FUNCTION_BLOCK ACMethodRouteBase EXTENDS ACMethodBase IMPLEMENTS IACMethodRouteBase
VAR_INPUT
END_VAR
VAR_OUTPUT
END_VAR
VAR
END_VAR
VAR PERSISTENT
	_Route : PARoute;
END_VAR

METHOD PUBLIC AssignRoute : BOOL
VAR_INPUT
	iAssignWithFunction : IPAProcessFunction;
END_VAR
VAR
	i : INT;
	iControlModule : IPAControlModule;
END_VAR
IF NOT _Route._IsResolved THEN
	AssignRoute := FALSE;
	RETURN;
END_IF

// TODO: Wegwechsel einbauen bzw. aktualsiierung der Route vom Client aus?

// Prüfe zuerst ob alle Stuerungsmodule nicht belegt sind
FOR i:=1 TO GCL.cRouteItemMAX BY 1
  DO    
  	IF _Route._Items[i] <> 0 THEN
		IF __QUERYINTERFACE(_Route._Items[i].Source.Parent, iControlModule) THEN
			IF iControlModule.AllocatedByWay THEN
				AssignRoute := FALSE;
				RETURN;				
			END_IF
		END_IF
		IF __QUERYINTERFACE(_Route._Items[i].Target.Parent, iControlModule) THEN
			IF iControlModule.AllocatedByWay THEN
				AssignRoute := FALSE;
				RETURN;				
			END_IF
		END_IF
	END_IF
  	_Route._Items[i] := 0;
END_FOR;

// Setze Belegung durch diese Funktion
FOR i:=1 TO GCL.cRouteItemMAX BY 1
  DO    
  	IF _Route._Items[i] <> 0 THEN
		IF __QUERYINTERFACE(_Route._Items[i].Source.Parent, iControlModule) THEN
			iControlModule.AllocatedByFunction := iAssignWithFunction;
		END_IF
		IF __QUERYINTERFACE(_Route._Items[i].Target.Parent, iControlModule) THEN
			iControlModule.AllocatedByFunction := iAssignWithFunction;
		END_IF
		_Route._Items[i].AllocatedByFunction := iAssignWithFunction;
	END_IF
END_FOR;
_Route._IsAssigned := TRUE;
END_METHOD

PROPERTY PUBLIC FirstCModuleInRoute : IPAControlModule
GET
VAR
	i : INT;
	iControlModule : IPAControlModule;
END_VAR
FOR i:=1 TO GCL.cRouteItemMAX BY 1
  DO    
  	IF _Route._Items[i] <> 0 THEN
		IF __QUERYINTERFACE(_Route._Items[i].Source.Parent, iControlModule) THEN
			FirstCModuleInRoute := iControlModule;
			RETURN;
		END_IF
	END_IF
END_FOR;
FirstCModuleInRoute := 0;
END_GET
END_PROPERTY

PROPERTY PUBLIC LastCModuleInRoute : IPAControlModule
GET
VAR
	i : INT;
	iControlModule : IPAControlModule;
	iLastCModule : IPAControlModule;
END_VAR
iLastCModule := 0;
FOR i:=1 TO GCL.cRouteItemMAX BY 1
  DO    
  	IF _Route._Items[i] <> 0 THEN
		IF __QUERYINTERFACE(_Route._Items[i].Target.Parent, iControlModule) THEN
			iLastCModule := iControlModule;
			RETURN;
		END_IF
	ELSE
		EXIT;
	END_IF
END_FOR;
LastCModuleInRoute := iLastCModule;
END_GET
END_PROPERTY

METHOD PUBLIC ResetRoute
VAR_INPUT
END_VAR
VAR
	i : INT;
	iControlModule : IPAControlModule;
END_VAR
IF NOT _Route._IsResolved AND NOT _Route._IsAssigned THEN
	RETURN;
END_IF
FOR i:=1 TO GCL.cRouteItemMAX BY 1
  DO    
  	// Lösche Wegebelegung auf den Steuerungsmodulen
  	IF  _Route._Items[i] <> 0 THEN
		IF __QUERYINTERFACE(_Route._Items[i].Source.Parent, iControlModule) THEN
			iControlModule.AllocatedByFunction := 0;
		END_IF
		IF __QUERYINTERFACE(_Route._Items[i].Target.Parent, iControlModule) THEN
			iControlModule.AllocatedByFunction := 0;
		END_IF
	END_IF
  	_Route._Items[i] := 0;
END_FOR;
_Route._IsResolved := FALSE;
_Route._IsAssigned := FALSE;
END_METHOD

METHOD PUBLIC ResolveRoutePointers : BOOL
VAR_INPUT
	routeToResolve : PARoutePointers;	
	parentComp : IACComponent;
END_VAR
VAR
	i: INT;
	pEdge : IACEdge;
	pEdgeToTest : IACObject;
END_VAR
FOR i:=1 TO GCL.cRouteItemMAX BY 1
  DO
  	_Route._Items[i] := 0;
	IF routeToResolve._InstanceID[i] = 0 THEN
		CONTINUE;
	END_IF
	pEdgeToTest := parentComp.FindObjectByID(routeToResolve._InstanceID[i]);
	IF pEdgeToTest = 0 AND __QUERYINTERFACE(pEdgeToTest, pEdge) THEN
		_Route._Items[i] := pEdge;		
	END_IF
END_FOR;
_Route._IsResolved := TRUE;
END_METHOD

PROPERTY PUBLIC Route : PARoute
GET
Route := _Route;
END_GET
END_PROPERTY

END_FUNCTION_BLOCK

(* stored: Version 1.1.0.1, ProductVersion 3.1.4022.7
   POU ACMethodRouteBase: Id {f92ea2b6-0103-4083-9ec7-d643bb944132}, SpecialFunc None
   Method AssignRoute: Id {03406dd0-2b2c-455a-a85a-47dc4bd5e337}
   Property FirstCModuleInRoute: Id {27162ce5-5620-431d-b7a8-f2b257fbb57d}
   Get Get: Id {d437d142-8ff9-4378-b40e-0aa4bb72caa1}
   Property LastCModuleInRoute: Id {6fd6225f-b074-457f-988b-c05b459db755}
   Get Get: Id {3a094643-31f2-41b1-9515-bcd93e03adb1}
   Method ResetRoute: Id {33fe7a1c-00bb-4339-b838-2c6e06cd15dc}
   Method ResolveRoutePointers: Id {75300ac9-c793-451f-9707-ec23dbc9607a}
   Property Route: Id {f648304f-e6e6-4301-8fc7-f6bcc1c05516}
   Get Get: Id {1cfee147-c5a3-411c-800f-29184951d6d6} *)
